(* IEC 61131-3 sources: Palletizer_Control_with_Automation_Studio/Palletizer/Logical/Libraries/Signal_lib, 3 files *)

(* ---- SignalManagement_FB.st ---- *)
(* TODO: Add your comment here *)
FUNCTION_BLOCK SignalManagement_FB

	CASE OperationType OF
		START_CONFIGURATION:  (* Reset signals counts *)
			NumberOfAlarms := 0;
			NumberOfAnomalies := 0;
			NumberOfWarnings := 0;
			NumberOfInformation := 0;
			ResetEnable := FALSE;
		CONFIGURATION:
			(* counting signals *)
			CASE SignalType AND SIGNAL_TYPE_MASK OF
				ALARM:
					NumberOfAlarms := NumberOfAlarms + 1;
				ANOMALY:
					NumberOfAnomalies := NumberOfAnomalies + 1;
				WARNING:
					NumberOfWarnings := NumberOfWarnings + 1;
				INFORMATION:
					NumberOfInformation := NumberOfInformation + 1;
			END_CASE
		START_GENERATION:
			(* Prepare for generation *)
			ResetEnable := FALSE;
			SignalOutputs := NONE;
			ResetActivation := Reset AND NOT ResetOld;
			ResetOld := Reset;
			AuxResetActivation := KeyReset AND NOT KeyResetOld;
			KeyResetOld:= KeyReset;
			LogFile := '';
			MainMessage := '';

		GENERATION:
			CASE SignalType AND SIGNAL_TYPE_MASK OF
				ALARM:
					Index := NumberOfActiveAlarms;
					BaseIndex := 0;
					Condition := TRUE;
				ANOMALY:
					Index := NumberOfActiveAnomalies;
					BaseIndex := NumberOfAlarms;
					Condition := TRUE;
				WARNING:
					Index := NumberOfActiveWarning;
					BaseIndex := NumberOfAlarms + NumberOfAnomalies;
					Condition := FALSE;
				INFORMATION:
					Index := NumberOfActiveInformation;
					BaseIndex := NumberOfAlarms + NumberOfAnomalies + NumberOfWarnings;
					Condition := FALSE;
			END_CASE
			IF ActivationSignal AND NOT Signals[SignalCode] THEN
				Signals[SignalCode] := TRUE;
				Index := Index + 1;
				ActiveSignalCodes[BaseIndex + Index] := SignalCode;

				IF (SignalType AND SIGNAL_LOG_MASK) = DISPLAY_LOG THEN
					LogBuffer[SignalCode] := InputString;
				END_IF

			END_IF
			IF Condition AND Signals[SignalCode] AND NOT ActivationSignal AND (ActiveSignalCodes[BaseIndex + 1] = SignalCode) THEN
				ResetEnable := TRUE;
			END_IF

			IF (ResetActivation OR NOT Condition) AND Signals[SignalCode] AND NOT ActivationSignal AND (ActiveSignalCodes[BaseIndex + 1] = SignalCode) THEN
				Signals[SignalCode] := FALSE;
				FOR i := 2 TO Index DO
					ActiveSignalCodes[BaseIndex + i-1] := ActiveSignalCodes[BaseIndex + i];
				END_FOR;
				ActiveSignalCodes[BaseIndex + Index] := 0;
				Index :=  Index - 1;
				ResetActivation := FALSE; (* COMMENT THIS LINE TO GO BACK TO CUMULATIVE RESET *)

				IF (SignalType AND SIGNAL_LOG_MASK) = DISPLAY_LOG THEN
					LogBuffer[SignalCode] := ' ';
				END_IF

			END_IF
			CASE SignalType AND SIGNAL_TYPE_MASK OF
				ALARM:
					NumberOfActiveAlarms := Index;
				ANOMALY:
					NumberOfActiveAnomalies := Index;
				WARNING:
					NumberOfActiveWarning := Index;
				INFORMATION:
					NumberOfActiveInformation := Index;
			END_CASE
			IF Signals[SignalCode] THEN
				SignalOutputs := SignalOutputs OR SignalOutput;
			END_IF

		MESSAGES_GENERATION:

			LogFile := ' ';
			// ALARMS messages creation
			BaseIndex := 0;
			FOR i := 1 TO NumberOfActiveAlarms DO
				IF LogBuffer[ActiveSignalCodes[BaseIndex + i]] <> '' THEN
					LogFile := CONCAT(CONCAT(LogFile, CONCAT('ALARM : ',LogBuffer[ActiveSignalCodes[BaseIndex + i]])), ' \n ');
				END_IF
			END_FOR;

			// ANOMALIES messages creation
			BaseIndex := NumberOfAlarms;
			FOR i := 1 TO NumberOfActiveAnomalies DO
				IF LogBuffer[ActiveSignalCodes[BaseIndex + i]] <> '' THEN
					LogFile := CONCAT(CONCAT(LogFile,CONCAT('ANOMALY : ',LogBuffer[ActiveSignalCodes[BaseIndex + i]])), ' \n ');
				END_IF

			END_FOR;

			// WARNING messages creation
			BaseIndex := NumberOfAlarms + NumberOfAnomalies;
			FOR i := 1 TO NumberOfActiveWarning DO
				IF LogBuffer[ActiveSignalCodes[BaseIndex + i]] <> '' THEN
					LogFile := CONCAT(CONCAT(LogFile , CONCAT('WARNING : ',LogBuffer[ActiveSignalCodes[BaseIndex + i]])), ' \n ');
				END_IF
			END_FOR;

			// WARNING messages creation
			BaseIndex := NumberOfAlarms + NumberOfAnomalies + NumberOfWarnings;
			FOR i := 1 TO NumberOfActiveInformation DO
				IF LogBuffer[ActiveSignalCodes[BaseIndex + i]] <> '' THEN
					LogFile := CONCAT(CONCAT(LogFile , CONCAT('INFORMATION : ',LogBuffer[ActiveSignalCodes[BaseIndex + i]])), ' \n ');
				END_IF
			END_FOR;

			MainMessage := '';
			IF NumberOfActiveAlarms <> 0 THEN
				MainMessage := LogBuffer[ActiveSignalCodes[1]];
			ELSIF NumberOfActiveAnomalies <> 0 THEN
				MainMessage := LogBuffer[ActiveSignalCodes[NumberOfAlarms + 1]];
			ELSIF NumberOfActiveWarning <> 0 THEN
				MainMessage := LogBuffer[ActiveSignalCodes[NumberOfAlarms + NumberOfAnomalies + 1]];
			ELSIF NumberOfActiveInformation <> 0 THEN
				MainMessage := LogBuffer[ActiveSignalCodes[NumberOfAlarms + NumberOfAnomalies + NumberOfWarnings + 1]];
			END_IF

	END_CASE

END_FUNCTION_BLOCK

(* ---- Signal_lib.fun ---- *)
{REDUND_ERROR} FUNCTION_BLOCK SignalManagement_FB (*TODO: Add your comment here*) (*$GROUP=User,$CAT=User,$GROUPICON=User.png,$CATICON=User.png*)
	VAR_INPUT
		OperationType : INT;
		SignalType : INT; (* bit configuration for the signal*)
		Reset : BOOL;
		KeyReset : BOOL;
		SignalOutput : DWORD; (* Output of the Signal if active*)
		ActivationSignal : {REDUND_UNREPLICABLE} BOOL;
		SignalCode : INT; (* Is the signal number in the priority list*)
		InputString : STRING[80];
	END_VAR
	VAR_OUTPUT
		MainMessage : STRING[30];
		LogFile : STRING[3000];
		SignalOutputs : DWORD; (*Output Signal codification*)
	END_VAR
	VAR
		LogBuffer : ARRAY[1..100] OF STRING[30];
		NumberOfAlarms : INT; (*Counters*)
		NumberOfAnomalies : INT;
		NumberOfWarnings : INT;
		NumberOfInformation : INT; (*Counters for Active Signals*)
		NumberOfActiveAlarms : INT;
		NumberOfActiveAnomalies : INT;
		NumberOfActiveWarning : INT;
		NumberOfActiveInformation : INT; (*Reset Management*)
	END_VAR
	VAR_OUTPUT
		ResetEnable : BOOL;
	END_VAR
	VAR
		ResetActivation : BOOL;
		AuxResetActivation : BOOL;
		Signals : ARRAY[1..100] OF BOOL; (*Signals management*)
		ActiveSignalCodes : ARRAY[1..100] OF INT;
		ResetOld : BOOL; (*Auxiliary variable*)
		KeyResetOld : BOOL;
		Index : INT;
		BaseIndex : INT;
		Condition : BOOL;
		i : INT;
	END_VAR
END_FUNCTION_BLOCK

(* ---- Constants.var ---- *)
(*OUTPUTS*)
VAR CONSTANT
	NONE : DWORD := 16#0000;
	EMERGENCY_STOP : DWORD := 16#0001;
	ON_PHASE_STOP : DWORD := 16#0010;
	IMMEDIATE_STOP : DWORD := 16#0100; (*Operation types for the Signal Manager*)
	START_CONFIGURATION : USINT := 1;
	CONFIGURATION : USINT := 2;
	START_GENERATION : USINT := 3;
	MESSAGES_GENERATION : USINT := 5;
	GENERATION : USINT := 4; (*SignalCode bitmap*)
	INFORMATION : USINT := 1;
	ANOMALY : USINT := 2;
	WARNING : USINT := 3;
	ALARM : USINT := 4; (*masks for the SiglaCode*)
	DISPLAY_LOG : USINT := 8;
	SIGNAL_TYPE_MASK : USINT := 7;
	SIGNAL_LOG_MASK : USINT := 8;
END_VAR
